// Mitsubishi GX Works2 project: 0625(MOV)   PLC: Q02/Q02H

PROGRAM MAIN
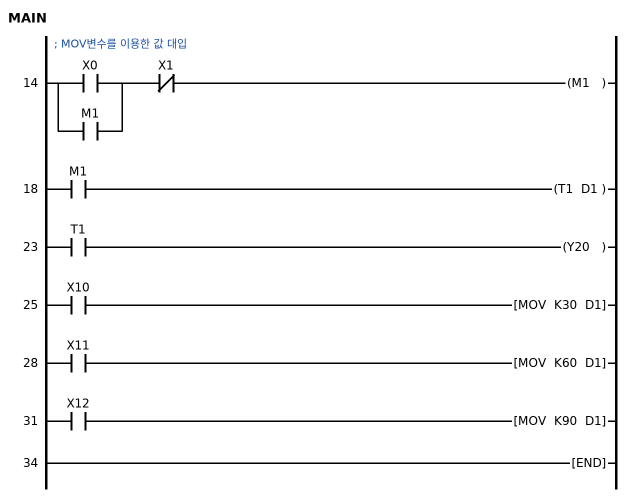
; MOV변수를 이용한 값 대입
14    LD      X0
      OR      M1
      ANI     X1
      OUT     M1
18    LD      M1
      OUT     T1 D1
23    LD      T1
      OUT     Y20
25    LD      X10
      MOV     K30 D1
28    LD      X11
      MOV     K60 D1
31    LD      X12
      MOV     K90 D1
34    END
END_PROGRAM
